% RSLogix 500 project COMPARA.RSS, saved by version 8.40.00.08 %
PROJECT "COMPARA"    % processor: MicroLogix 1500 %

PROGRAM FILES
  LAD 2   3 rungs

DATA FILES
  O0 OUTPUT  14 elements
  I1 INPUT  26 elements
  S2 STATUS  66 elements
  B3 BINARY  1 elements
  T4 TIMER  1 elements
  C5 COUNTER  1 elements
  R6 CONTROL  1 elements
  N7 INTEGER  1 elements
  F8 FLOAT  1 elements

LADDER 2
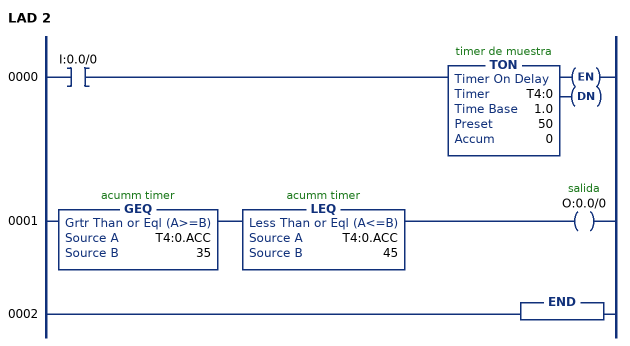
% Rung: 0 %
SOR XIC I:0.0/0 TON T4:0 1.0 50 0 EOR
%   T4:0  "timer de muestra" %
% Rung: 1 %
SOR GEQ T4:0.ACC 35 LEQ T4:0.ACC 45 OTE O:0.0/0 EOR
%   T4:0.ACC  "acumm timer" %
%   O:0.0/0  "salida" %
% Rung: 2 %
SOR END EOR

OTHER DOCUMENTED ADDRESSES
  C5:0  "Contador muestra"
  C5:0.ACC  "Accum contador"

DATA TABLE (non-zero values as saved)
DATA T4
% .PRE .ACC %
% T4:0 % 50 0
DATA C5
% .PRE .ACC %
% C5:0 % 25 0
